{attribute 'qualified_only'}
TYPE E_LubricationMode :
(
	TimeBased,
	DistanceBased,
	Continous
);
END_TYPE

(* stored: Version 1.1.0.1, ProductVersion 3.1.4024.12
   DUT E_LubricationMode: Id {377c692d-3be3-43aa-b41d-3f9425f56c5b} *)
